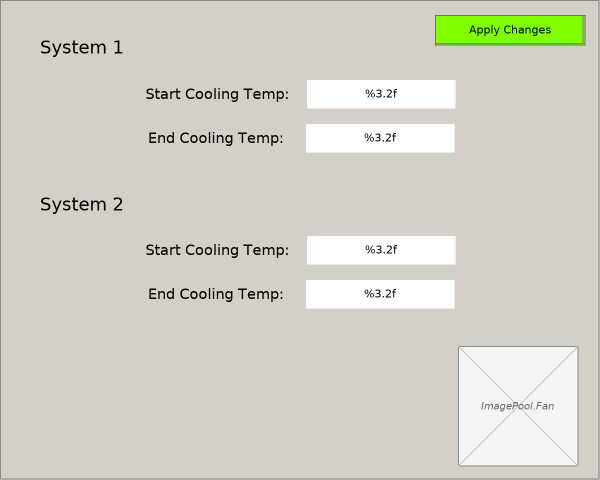
VISUALIZATION vCooling  // 600x480
    Label (28,35 108x25), "System 1"
    Label (28,192 108x25), "System 2"
    Button (435,15 150x30), "Apply Changes"
        OnMouseClick: execute { MAIN.bSetPerData:=true; }
    Textfield (305,279 150x30), "%3.2f", text variable: ACTION2.rEndCoolingTemp
        OnMouseClick: write the text variable via Default
    Textfield (306,235 150x30), "%3.2f", text variable: ACTION2.rStartCoolingTemp
        OnMouseClick: write the text variable via Default
    Textfield (305,123 150x30), "%3.2f", text variable: ACTION1.rEndCoolingTemp
        OnMouseClick: write the text variable via Default
    Label (137,123 158x30), "End Cooling Temp:"
    Textfield (306,79 150x30), "%3.2f", text variable: ACTION1.rStartCoolingTemp
        OnMouseClick: write the text variable via Default
    Label (137,79 161x30), "Start Cooling Temp:"
    Image (458,346 120x120), image: ImagePool.Fan
    Label (137,235 161x30), "Start Cooling Temp:"
    Label (137,279 158x30), "End Cooling Temp:"
END_VISUALIZATION

(* stored: Version 1.1.0.1, ProductVersion 3.1.4024.12
   Visu vCooling: Id {c1913d97-3c20-4046-972c-8e18a79c5b62} *)
